PROGRAM MAIN
VAR
END_VAR

GVL_Data.stRecipe.eMachineType:=E_MachineType.RH069;
P_System();//系统程序
P_Alarm();// 报警程序
P_Device();// 外围装置
P_Station();// 工站流程

END_PROGRAM

(* stored: Version 1.1.0.1, ProductVersion 3.1.4024.3
   POU MAIN: Id {9f111226-449a-4e9b-8be2-b4171f48ff56}, SpecialFunc None *)
